Staubli VAL3: Trasladar.dtx

bool bTraslada
bool bFin
bool bPiezaPreparada
bool bTermina
jointRx jHome
public mdesc mNomSpeed = {leave=25, reach=25}
mdesc mVelAprox = {accel=25, vel=50, decel=25, blend=off}
num nPendientes
num nSolicitadas = 2
pointRx pEntrada = {x=-415, y=250, z=-265, ry=-180, shoulder=lefty, elbow=epositive, wrist=wpositive, fatherId=world[0]}
pointRx pEspera = {x=-415, y=250, z=-215, rx=-180, ry=-7.016709E-15, rz=-180, shoulder=lefty, elbow=epositive, wrist=wpositive, fatherId=world[0]}
pointRx pSalida = {x=-415, z=-210, ry=-180, fatherId=world[0]}
string sMensaje
tool tEyector = {z=22, fatherId=flange[0], ioLink=valve1, ioOpen=1, ioClose=1}
trsf trAprox = {z=-50}
